Staubli VAL3: sampleChangerV4.dtx

bool taskIsDone
dio switchGripper = {link=valve1}
jointRx binPosition = {j1=59.154914, j2=15.287075, j3=144.068937, j4=0.00349, j5=20.640131, j6=239.148927}
jointRx currentPickPosJ = {j1=24.086468, j2=103.725715, j3=36.339858, j4=-71.090092, j5=105.162663, j6=322.602811}
jointRx currentSamPosJ = {j1=64.5166, j2=21.7725, j3=135.395, j4=0.005, j5=22.8226, j6=244.506}
jointRx gatePosition = {j1=53.332436, j2=31.008098, j3=108.023775, j4=-0.035914, j5=40.963114, j6=323.353672}
jointRx homePosition = {j1=64.5166, j2=21.7725, j3=135.395, j4=0.005, j5=22.8226, j6=244.506}
jointRx parkingPosition = {j1=20.774519, j2=86.925335, j3=58.285959, j4=-72.455135, j5=101.349332, j6=295.989419}
jointRx spinnerPosition = {j1=24.224814, j2=103.543996, j3=36.557875, j4=-70.964584, j5=105.220885, j6=322.664695}
jointRx zeroPosition = {j1=88.745927, j2=-26.51301, j3=117.695598, j4=-0.539561, j5=89.308877, j6=269.442332}
mdesc mFastMov = {blend=off}
mdesc mNomSpeed = {accel=2.25, vel=15, decel=2.25}
num coords[2]
  [0] = 4
  [1] = 9
num numMessage[32]
num numSpeed = 5
num numXarray = 1
num numXold
num numYarray = 1
num numYold
pointRx currentPickPos = {x=982.652852, y=394.034002, z=-652.657917, rx=90.013165, ry=0.023145, rz=89.994895, shoulder=lefty, elbow=epositive, wrist=wpositive, fatherId=world[0]}
pointRx currentSamPos = {x=188.431145, y=511.898865, z=-95.729646, rx=-179.992666, ry=0.001448, rz=-0.004557, shoulder=lefty, elbow=epositive, wrist=wpositive, fatherId=world[0]}
sio sioASCII[2]
  [0] = {link=Socket\tan}
  [1] = {link=Socket\tan}
